INTERFACE I_Clear

METHOD Clear : I_SetNumber
END_METHOD

END_INTERFACE

(* stored: Version 1.1.0.1, ProductVersion 3.1.4024.12
   Itf I_Clear: Id {83be75c4-62a3-4d02-8eb0-dde04a84ab35}
   Method Clear: Id {195c8fc3-ce62-471f-8dec-0cc2a3f7ae6b} *)
